KUKA KRL data list: ps_p13060r5_stb_resp_c2.dat

&ACCESS RVO
&REL 19
&COMMENT C2 Respot STB
&PARAM DISKPATH = KRC:\R1\Program
DEFDAT  ps_p13060r5_stb_resp_c2
;FOLD EXTERNAL DECLARATIONS;%{PE}%MKUKATPBASIS,%CEXT,%VCOMMON,%P
;FOLD GRIPPERTECH EXT
EXT  H50 (INT  :IN,INT  :IN,INT  :IN,GRP_TYP  :IN )
;ENDFOLD (GRIPPERTECH EXT)
;FOLD SPOTTECH EXT
EXT  USERSPOT (S_COMMAND  :IN,SPOT_TYPE  :IN )
;ENDFOLD (SPOTTECH EXT)
;FOLD BASISTECH EXT;%{PE}%MKUKATPBASIS,%CEXT,%VEXT,%P
EXT  BAS (BAS_COMMAND  :IN,REAL  :IN )
DECL INT SUCCESS
;ENDFOLD (BASISTECH EXT)
;FOLD USER EXT;%{E}%MKUKATPUSER,%CEXT,%VEXT,%P
;Make your modifications here

;ENDFOLD (USER EXT)
;ENDFOLD (EXTERNAL DECLARATIONS)

;# ============ START PATH : swp_p13060r5_stb_resp_c2 =============
DECL FDAT Fp108={TOOL_NO 3,BASE_NO 1,IPO_FRAME #BASE,POINT2[] " "}
DECL PDAT PP_OLP2={VEL 100.0,ACC 100.0,APO_DIST 100.0,APO_MODE #CDIS}
DECL E6POS Xp108={X 827.567993,Y 431.752991,Z 2345.34912,A -125.237503,B 71.8876038,C -48.1716003,S 2,T 42}
DECL FDAT Fp109={TOOL_NO 3,BASE_NO 1,IPO_FRAME #BASE,POINT2[] " "}
DECL PDAT PP_OLP3={VEL 100.0,ACC 100.0,APO_DIST 100.0,APO_MODE #CDIS}
DECL E6POS Xp109={X 1037.08301,Y 431.752991,Z 1323.84497,A -35.7363014,B 64.2305984,C 45.5069008,S 2,T 42}
DECL FDAT Fp110={TOOL_NO 3,BASE_NO 1,IPO_FRAME #BASE,POINT2[] " "}
DECL PDAT PP_OLP4={VEL 100.0,ACC 100.0,APO_DIST 100.0,APO_MODE #CDIS}
DECL E6POS Xp110={X 1446.06604,Y 997.797974,Z 625.557922,A 43.6373405,B 73.7974472,C 136.977997,S 6,T 56,E1 0.0,E2 0.0,E3 0.0,E4 0.0,E5 0.0,E6 0.0}
DECL FDAT Fp112={TOOL_NO 3,BASE_NO 1,IPO_FRAME #BASE,POINT2[] " "}
DECL PDAT PP_OLP6={VEL 100.0,ACC 100.0,APO_DIST 100.0,APO_MODE #CDIS}
DECL E6POS Xp112={X 1490.95496,Y 1047.58301,Z 618.734924,A 51.0465202,B 81.7684631,C 154.884903,S 6,T 56,E1 0.0,E2 0.0,E3 0.0,E4 0.0,E5 0.0,E6 0.0}
DECL FDAT Fp113={TOOL_NO 3,BASE_NO 1,IPO_FRAME #BASE,POINT2[] " "}
DECL PDAT PP_OLP7={VEL 100.0,ACC 100.0,APO_DIST 100.0,APO_MODE #CDIS}
DECL E6POS Xp113={X 1494.36499,Y 1136.25806,Z 483.507904,A 36.9966698,B 83.4788284,C 134.325394,S 6,T 56,E1 0.0,E2 0.0,E3 0.0,E4 0.0,E5 0.0,E6 0.0}
DECL FDAT Fswp_60_4492={TOOL_NO 3,BASE_NO 1,IPO_FRAME #BASE,POINT2[] " "}
DECL PDAT PP_OLP9={VEL 100.0,ACC 100.0,APO_DIST 0.0}
DECL SPOT_TYPE SS_OLP1={GUN 3,PAIR #FIRST,RETR #CLO,CLO_TM 0,PGNO1 1,PRESS1 1.0,PGNO2 0,PRESS2 0.0}
DECL E6POS Xswp_60_4492={X 1524.54602,Y 1133.35205,Z 403.493988,A -0.563865423,B 81.9408188,C 90.5450287,S 6,T 56,E1 0.0,E2 0.0,E3 0.0,E4 0.0,E5 0.0,E6 0.0}
DECL FDAT Fswp_60_4490={TOOL_NO 3,BASE_NO 1,IPO_FRAME #BASE,POINT2[] " "}
DECL PDAT PP_OLP10={VEL 100.0,ACC 100.0,APO_DIST 0.0}
DECL SPOT_TYPE SS_OLP2={GUN 3,PAIR #FIRST,RETR #CLO,CLO_TM 0,PGNO1 1,PRESS1 1.0,PGNO2 0,PRESS2 0.0}
DECL E6POS Xswp_60_4490={X 1542.60596,Y 1134.66602,Z 422.517792,A -0.0879144073,B 77.980423,C 91.234787,S 6,T 56,E1 0.0,E2 0.0,E3 0.0,E4 0.0,E5 0.0,E6 0.0}
DECL FDAT Fp115={TOOL_NO 3,BASE_NO 1,IPO_FRAME #BASE,POINT2[] " "}
DECL PDAT PP_OLP11={VEL 100.0,ACC 100.0,APO_DIST 100.0,APO_MODE #CDIS}
DECL E6POS Xp115={X 1542.29297,Y 1134.60205,Z 455.016602,A -0.0876709968,B 77.9804077,C 91.2347717,S 6,T 56,E1 0.0,E2 0.0,E3 0.0,E4 0.0,E5 0.0,E6 0.0}
DECL FDAT Fswp_60_4488={TOOL_NO 3,BASE_NO 1,IPO_FRAME #BASE,POINT2[] " ",TQ_STATE FALSE}
DECL PDAT PP_OLP12={VEL 100.0,ACC 100.0,APO_DIST 0.0}
DECL SPOT_TYPE SS_OLP3={GUN 3,PAIR #FIRST,RETR #CLO,CLO_TM 0,PGNO1 1,PRESS1 1.0,PGNO2 0,PRESS2 0.0}
DECL E6POS Xswp_60_4488={X 1568.30103,Y 1134.96399,Z 453.733185,A 0.514110625,B 75.6271667,C 91.8389893,S 6,T 56,E1 0.0,E2 0.0,E3 0.0,E4 0.0,E5 0.0,E6 0.0}
DECL FDAT Fswp_60_4486={TOOL_NO 3,BASE_NO 1,IPO_FRAME #BASE,POINT2[] " "}
DECL PDAT PP_OLP13={VEL 100.0,ACC 100.0,APO_DIST 0.0}
DECL SPOT_TYPE SS_OLP4={GUN 3,PAIR #FIRST,RETR #CLO,CLO_TM 0,PGNO1 1,PRESS1 1.0,PGNO2 0,PRESS2 0.0}
DECL E6POS Xswp_60_4486={X 1597.06494,Y 1131.53796,Z 456.258087,A 0.623319328,B 71.0001373,C 91.9330673,S 6,T 24,E1 0.0,E2 0.0,E3 0.0,E4 0.0,E5 0.0,E6 0.0}
DECL FDAT Fp117={TOOL_NO 3,BASE_NO 1,IPO_FRAME #BASE,POINT2[] " "}
DECL E6POS Xp117={X 1518.06201,Y 1123.82605,Z 532.922424,A 23.5638008,B 79.3738937,C 119.158897,S 6,T 56,E1 0.0,E2 0.0,E3 0.0,E4 0.0,E5 0.0,E6 0.0}
DECL FDAT Fp118={TOOL_NO 3,BASE_NO 1,IPO_FRAME #BASE,POINT2[] " "}
DECL PDAT PP_OLP16={VEL 100.0,ACC 100.0,APO_DIST 100.0,APO_MODE #CDIS}
DECL E6POS Xp118={X 1495.46802,Y 1131.28406,Z 618.445679,A 51.6626511,B 81.6151733,C 150.156204,S 6,T 56,E1 0.0,E2 0.0,E3 0.0,E4 0.0,E5 0.0,E6 0.0}
DECL FDAT Fp119={TOOL_NO 3,BASE_NO 1,IPO_FRAME #BASE,POINT2[] " "}
DECL PDAT PP_OLP17={VEL 100.0,ACC 100.0,APO_DIST 100.0,APO_MODE #CDIS}
DECL E6POS Xp119={X 1491.46899,Y 1011.04199,Z 618.887817,A 51.6626511,B 81.6151733,C 150.156204,S 6,T 56,E1 0.0,E2 0.0,E3 0.0,E4 0.0,E5 0.0,E6 0.0}
DECL FDAT Fp121={TOOL_NO 3,BASE_NO 1,IPO_FRAME #BASE,POINT2[] " "}
DECL PDAT PP_OLP19={VEL 100.0,ACC 100.0,APO_DIST 100.0,APO_MODE #CDIS}
DECL E6POS Xp121={X 941.241272,Y -14.3455095,Z 1188.11304,A 0.321344793,B 55.8508301,C 1.17380595,S 6,T 51,E1 0.0,E2 0.0,E3 0.0,E4 0.0,E5 0.0,E6 0.0}
DECL FDAT Fp124={TOOL_NO 3,BASE_NO 1,IPO_FRAME #BASE,POINT2[] " "}
DECL PDAT PP_OLP22={VEL 100.0,ACC 100.0,APO_DIST 100.0,APO_MODE #CDIS}
DECL E6POS Xp124={X 1503.23901,Y -1033.73206,Z 643.593018,A -59.5746384,B 73.2440033,C -157.993195,S 6,T 17,E1 0.0,E2 0.0,E3 0.0,E4 0.0,E5 0.0,E6 0.0}
DECL FDAT Fp125={TOOL_NO 3,BASE_NO 1,IPO_FRAME #BASE,POINT2[] " "}
DECL PDAT PP_OLP23={VEL 100.0,ACC 100.0,APO_DIST 100.0,APO_MODE #CDIS}
DECL E6POS Xp125={X 1530.15796,Y -1124.66199,Z 618.227722,A -59.5806885,B 73.2442322,C -158.002304,S 6,T 17,E1 0.0,E2 0.0,E3 0.0,E4 0.0,E5 0.0,E6 0.0}
DECL FDAT Fp128={TOOL_NO 3,BASE_NO 1,IPO_FRAME #BASE,POINT2[] " "}
DECL PDAT PP_OLP26={VEL 100.0,ACC 100.0,APO_DIST 100.0,APO_MODE #CDIS}
DECL E6POS Xp128={X 1550.953,Y -1131.5,Z 478.679199,A 7.11577177,B 79.6360397,C -90.3111267,S 6,T 17,E1 0.0,E2 0.0,E3 0.0,E4 0.0,E5 0.0,E6 0.0}
DECL FDAT Fswp_60_4491={TOOL_NO 3,BASE_NO 1,IPO_FRAME #BASE,POINT2[] " "}
DECL PDAT PP_OLP27={VEL 100.0,ACC 100.0,APO_DIST 0.0}
DECL SPOT_TYPE SS_OLP5={GUN 3,PAIR #FIRST,RETR #CLO,CLO_TM 0,PGNO1 1,PRESS1 1.0,PGNO2 0,PRESS2 0.0}
DECL E6POS Xswp_60_4491={X 1556.48804,Y -1128.06299,Z 414.378113,A 7.11510181,B 79.6364594,C -90.3119965,S 6,T 17,E1 0.0,E2 0.0,E3 0.0,E4 0.0,E5 0.0,E6 0.0}
DECL FDAT Fswp_60_4489={TOOL_NO 3,BASE_NO 1,IPO_FRAME #BASE,POINT2[] " "}
DECL PDAT PP_OLP28={VEL 100.0,ACC 100.0,APO_DIST 0.0}
DECL SPOT_TYPE SS_OLP6={GUN 3,PAIR #FIRST,RETR #CLO,CLO_TM 0,PGNO1 1,PRESS1 1.0,PGNO2 0,PRESS2 0.0}
DECL E6POS Xswp_60_4489={X 1571.31006,Y -1127.97498,Z 435.016602,A 7.13421679,B 78.9879608,C -90.2929916,S 6,T 17,E1 0.0,E2 0.0,E3 0.0,E4 0.0,E5 0.0,E6 0.0}
DECL FDAT Fp129={TOOL_NO 3,BASE_NO 1,IPO_FRAME #BASE,POINT2[] " "}
DECL PDAT PP_OLP29={VEL 100.0,ACC 100.0,APO_DIST 100.0,APO_MODE #CDIS}
DECL E6POS Xp129={X 1568.74902,Y -1124.86597,Z 460.267303,A 4.05743599,B 78.2943268,C -92.4355164,S 6,T 17,E1 0.0,E2 0.0,E3 0.0,E4 0.0,E5 0.0,E6 0.0}
DECL FDAT Fswp_60_4487={TOOL_NO 3,BASE_NO 1,IPO_FRAME #BASE,POINT2[] " "}
DECL PDAT PP_OLP30={VEL 100.0,ACC 100.0,APO_DIST 0.0}
DECL SPOT_TYPE SS_OLP7={GUN 3,PAIR #FIRST,RETR #CLO,CLO_TM 0,PGNO1 1,PRESS1 1.0,PGNO2 0,PRESS2 0.0}
DECL E6POS Xswp_60_4487={X 1595.77295,Y -1126.99695,Z 462.391815,A 0.286340088,B 72.7262421,C -91.5810623,S 6,T 17,E1 0.0,E2 0.0,E3 0.0,E4 0.0,E5 0.0,E6 0.0}
DECL FDAT Fswp_60_4485={TOOL_NO 3,BASE_NO 1,IPO_FRAME #BASE,POINT2[] " "}
DECL PDAT PP_OLP31={VEL 100.0,ACC 100.0,APO_DIST 0.0}
DECL SPOT_TYPE SS_OLP8={GUN 3,PAIR #FIRST,RETR #CLO,CLO_TM 0,PGNO1 1,PRESS1 1.0,PGNO2 0,PRESS2 0.0}
DECL E6POS Xswp_60_4485={X 1618.53601,Y -1124.83496,Z 464.984985,A 1.588274,B 72.3667374,C -91.6739731,S 6,T 17,E1 0.0,E2 0.0,E3 0.0,E4 0.0,E5 0.0,E6 0.0}
DECL FDAT Fp130={TOOL_NO 3,BASE_NO 1,IPO_FRAME #BASE,POINT2[] " "}
DECL PDAT PP_OLP32={VEL 100.0,ACC 100.0,APO_DIST 100.0,APO_MODE #CDIS}
DECL E6POS Xp130={X 1565.98901,Y -1121.01099,Z 457.081299,A 1.79761195,B 76.434227,C -91.4393005,S 6,T 17,E1 0.0,E2 0.0,E3 0.0,E4 0.0,E5 0.0,E6 0.0}
DECL FDAT Fp131={TOOL_NO 3,BASE_NO 1,IPO_FRAME #BASE,POINT2[] " "}
DECL PDAT PP_OLP33={VEL 100.0,ACC 100.0,APO_DIST 100.0,APO_MODE #CDIS}
DECL E6POS Xp131={X 1569.81104,Y -1127.59998,Z 558.258423,A -15.1613102,B 74.2022018,C -113.335701,S 6,T 17,E1 0.0,E2 0.0,E3 0.0,E4 0.0,E5 0.0,E6 0.0}
DECL FDAT Fp134={TOOL_NO 3,BASE_NO 1,IPO_FRAME #BASE,POINT2[] " "}
DECL PDAT PP_OLP36={VEL 100.0,ACC 100.0,APO_DIST 100.0,APO_MODE #CDIS}
DECL E6POS Xp134={X 1522.56396,Y -1127.91394,Z 647.963196,A -59.0981293,B 76.7364502,C -158.186096,S 6,T 17,E1 0.0,E2 0.0,E3 0.0,E4 0.0,E5 0.0,E6 0.0}
DECL FDAT Fp135={TOOL_NO 3,BASE_NO 1,IPO_FRAME #BASE,POINT2[] " "}
DECL PDAT PP_OLP37={VEL 100.0,ACC 100.0,APO_DIST 100.0,APO_MODE #CDIS}
DECL E6POS Xp135={X 1513.45496,Y -1035.99902,Z 649.452026,A -52.8882599,B 75.6186371,C -152.715103,S 6,T 17,E1 0.0,E2 0.0,E3 0.0,E4 0.0,E5 0.0,E6 0.0}
DECL FDAT Fp137={TOOL_NO 3,BASE_NO 1,IPO_FRAME #BASE,POINT2[] " "}
DECL PDAT PP_OLP39={VEL 100.0,ACC 100.0,APO_DIST 100.0,APO_MODE #CDIS}
DECL E6POS Xp137={X 1520.76697,Y -991.889282,Z 650.228577,A -10.46768,B 80.2553711,C -117.978798,S 6,T 17,E1 0.0,E2 0.0,E3 0.0,E4 0.0,E5 0.0,E6 0.0}
DECL FDAT Fp139={TOOL_NO 3,BASE_NO 1,IPO_FRAME #BASE,POINT2[] " "}
DECL PDAT PP_OLP41={VEL 100.0,ACC 100.0,APO_DIST 0.0,APO_MODE #CDIS}
DECL E6POS Xp139={X 1281.24805,Y 309.811615,Z 1549.84204,A -76.818718,B 70.1210022,C 12.2677097,S 6,T 51,E1 0.0,E2 0.0,E3 0.0,E4 0.0,E5 0.0,E6 0.0}
DECL E6POS XP2={X 1496.05603,Y 1141.896,Z 618.40918,A 51.6626205,B 81.6152191,C 150.156296,S 6,T 56,E1 0.0,E2 0.0,E3 0.0,E4 0.0,E5 0.0,E6 0.0}
DECL FDAT FP2={TOOL_NO 3,BASE_NO 1,IPO_FRAME #BASE,POINT2[] " ",TQ_STATE FALSE}
DECL PDAT PPDAT2={VEL 100.0,ACC 100.0,APO_DIST 100.0}
DECL SPOT_SUGG_T LAST_SPOT={GUN[] "1                       ",RETR_CMD[] "#OPN                    ",CHOISE[] "#FIRST                  ",CLO_TM[] "0                       ",PGNO1[] "1                       ",PRESS1[] "0                       ",PGNO2[] "1                       ",PRESS2[] "0                       ",SPOT_PARAMS[] "NORMAL                  "}
DECL LDAT LCPDAT1={VEL 2.0,ACC 100.0,APO_DIST 100.0,APO_FAC 50.0,AXIS_VEL 100.0,AXIS_ACC 100.0,ORI_TYP #VAR,CIRC_TYP #BASE,JERK_FAC 50.0,GEAR_JERK 50.0,EXAX_IGN 0}
DECL E6POS XP3={X 964.991272,Y 470.910309,Z 2238.42407,A -112.884804,B 77.3876419,C -21.04006,S 6,T 51,E1 0.0,E2 0.0,E3 0.0,E4 0.0,E5 0.0,E6 0.0}
DECL FDAT FP3={TOOL_NO 3,BASE_NO 1,IPO_FRAME #BASE,POINT2[] " ",TQ_STATE FALSE}
DECL PDAT PPDAT4={VEL 100.0,ACC 100.0,APO_DIST 100.0,APO_MODE #CDIS}
DECL PDAT PPDAT6={VEL 100.0,ACC 100.0,APO_DIST 100.0,APO_MODE #CDIS}
DECL E6POS XP5={X 412.222412,Y 36.2786789,Z 3142.17407,A -0.471725702,B 79.3877869,C -1.30059099,S 2,T 3,E1 0.0,E2 0.0,E3 0.0,E4 0.0,E5 0.0,E6 0.0}
DECL FDAT FP5={TOOL_NO 3,BASE_NO 1,IPO_FRAME #BASE,POINT2[] " ",TQ_STATE FALSE}
DECL PDAT PPDAT7={VEL 100.0,ACC 100.0,APO_DIST 100.0,APO_MODE #CDIS}
DECL E6POS XP6={X 412.222687,Y 36.2649193,Z 3142.18701,A -0.471164703,B 79.3883667,C -1.30046999,S 2,T 3,E1 0.0,E2 0.0,E3 0.0,E4 0.0,E5 0.0,E6 0.0}
DECL FDAT FP6={TOOL_NO 3,BASE_NO 1,IPO_FRAME #BASE,POINT2[] " ",TQ_STATE FALSE}
DECL E6POS XP8={X 1617.97498,Y -1124.04895,Z 460.753204,A 1.59669602,B 72.3654633,C -91.6747665,S 6,T 17,E1 0.0,E2 0.0,E3 0.0,E4 0.0,E5 0.0,E6 0.0}
DECL FDAT FP8={TOOL_NO 3,BASE_NO 1,IPO_FRAME #BASE,POINT2[] " ",TQ_STATE FALSE}
DECL PDAT PPDAT9={VEL 100.0,ACC 100.0,APO_DIST 100.0,APO_MODE #CDIS}
DECL E6POS XP9={X 1482.32605,Y 1095.13501,Z 618.705322,A 51.2849197,B 81.6177216,C 152.702103,S 6,T 56,E1 0.0,E2 0.0,E3 0.0,E4 0.0,E5 0.0,E6 0.0}
DECL FDAT FP9={TOOL_NO 3,BASE_NO 1,IPO_FRAME #BASE,POINT2[] " ",TQ_STATE FALSE}
DECL PDAT PPDAT10={VEL 100.0,ACC 100.0,APO_DIST 5.0,APO_MODE #CDIS}
DECL E6POS XP10={X 1579.73401,Y 1128.98206,Z 457.32431,A 1.53559196,B 73.7870178,C 92.807518,S 6,T 24,E1 0.0,E2 0.0,E3 0.0,E4 0.0,E5 0.0,E6 0.0}
DECL FDAT FP10={TOOL_NO 3,BASE_NO 1,IPO_FRAME #BASE,POINT2[] " ",TQ_STATE FALSE}
DECL PDAT PPDAT11={VEL 100.0,ACC 100.0,APO_DIST 1.0,APO_MODE #CDIS}
DECL E6POS XP11={X 1551.53699,Y -1125.46704,Z 606.090576,A -34.0320587,B 75.3278503,C -132.666794,S 6,T 17,E1 0.0,E2 0.0,E3 0.0,E4 0.0,E5 0.0,E6 0.0}
DECL FDAT FP11={TOOL_NO 3,BASE_NO 1,IPO_FRAME #BASE,POINT2[] " ",TQ_STATE FALSE}
DECL PDAT PPDAT12={VEL 100.0,ACC 100.0,APO_DIST 2.0,APO_MODE #CDIS}
DECL E6POS XP12={X 1509.10803,Y 1126.86499,Z 440.299805,A 12.1597605,B 81.9712372,C 106.209702,S 6,T 56,E1 0.0,E2 0.0,E3 0.0,E4 0.0,E5 0.0,E6 0.0}
DECL FDAT FP12={TOOL_NO 3,BASE_NO 1,IPO_FRAME #BASE,POINT2[] " ",TQ_STATE FALSE}
DECL PDAT PPDAT13={VEL 100.0,ACC 100.0,APO_DIST 3.0,APO_MODE #CDIS}
DECL E6POS XP13={X 4596.02197,Y -991.739624,Z 4346.84521,A -37.4233208,B 45.9583511,C 122.2882,S 2,T 11,E1 0.0,E2 0.0,E3 0.0,E4 0.0,E5 0.0,E6 0.0}
DECL FDAT FP13={TOOL_NO 3,BASE_NO 1,IPO_FRAME #BASE,POINT2[] " ",TQ_STATE FALSE}
DECL PDAT PPDAT14={VEL 100.0,ACC 100.0,APO_DIST 5.0,APO_MODE #CDIS}
DECL E6POS XP14={X 2787.1731,Y -2269.57202,Z 4832.78076,A -92.1469727,B 17.6405602,C 131.842896,S 2,T 11,E1 0.0,E2 0.0,E3 0.0,E4 0.0,E5 0.0,E6 0.0}
DECL FDAT FP14={TOOL_NO 3,BASE_NO 1,IPO_FRAME #BASE,POINT2[] " ",TQ_STATE FALSE}
DECL PDAT PPDAT15={VEL 100.0,ACC 100.0,APO_DIST 5.0,APO_MODE #CDIS}
DECL E6POS XP15={X 2787.17212,Y -2269.573,Z 4832.77783,A -92.1469727,B 17.6406403,C 131.842896,S 2,T 11,E1 0.0,E2 0.0,E3 0.0,E4 0.0,E5 0.0,E6 0.0}
DECL FDAT FP15={TOOL_NO 3,BASE_NO 1,IPO_FRAME #BASE,POINT2[] " ",TQ_STATE FALSE}
DECL PDAT PPDAT16={VEL 100.0,ACC 100.0,APO_DIST 100.0,APO_MODE #CDIS}
DECL PDAT PPDAT0={VEL 100.0,ACC 100.0,APO_DIST 5.0,APO_MODE #CDIS}
DECL E6POS XP0={X 4486.14795,Y -1238.07104,Z 4489.45801,A -42.8202209,B 37.5040016,C 125.268799,S 2,T 11,E1 0.0,E2 0.0,E3 0.0,E4 0.0,E5 0.0,E6 0.0}
DECL FDAT FP0={TOOL_NO 3,BASE_NO 1,IPO_FRAME #BASE,POINT2[] " ",TQ_STATE FALSE}
ENDDAT
